// Mitsubishi GX Works2 project: FX2   PLC: FX2/FX2C

PROGRAM MAIN
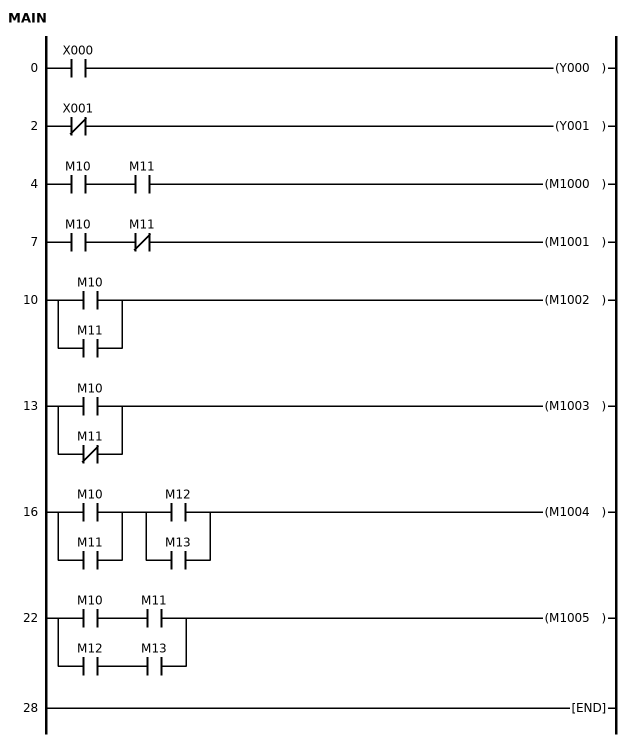
0     LD      X000
      OUT     Y000
2     LDI     X001
      OUT     Y001
4     LD      M10
      AND     M11
      OUT     M1000
7     LD      M10
      ANI     M11
      OUT     M1001
10    LD      M10
      OR      M11
      OUT     M1002
13    LD      M10
      ORI     M11
      OUT     M1003
16    LD      M10
      OR      M11
      LD      M12
      OR      M13
      ANB
      OUT     M1004
22    LD      M10
      AND     M11
      LD      M12
      AND     M13
      ORB
      OUT     M1005
28    END
END_PROGRAM
